{attribute 'qualified_only'}
VAR_GLOBAL
		Button : BOOL;     (* Input voor de knop *)
   		Lamp   : BOOL;     (* Output voor de lamp *)
END_VAR

(* stored: Version 1.1.0.1, ProductVersion 3.1.4024.12
   GVL GVL_Carbid: Id {8d2a7e60-294b-41ef-945d-fbc277f02d31} *)
